{attribute 'qualified_only'}
VAR_GLOBAL
	Variable1:REAL;
	id:GUID;
END_VAR

(* stored: Version 1.1.0.1, ProductVersion 3.1.4024.9
   GVL DB: Id {9653628f-efdc-46ab-863c-cf454af8c46d} *)
